INTERFACE I_EventReactionTcEvents EXTENDS I_EventReaction

METHOD GetHighestActiveEventSeverity : TcEventSeverity
END_METHOD

END_INTERFACE

(* stored: Version 1.1.0.1, ProductVersion 3.1.4026.18
   Itf I_EventReactionTcEvents: Id {9ba85094-bdcc-4410-92fb-9d3383e4ff12}
   Method GetHighestActiveEventSeverity: Id {472bb527-7b81-40a7-b14e-172cd6ea18e1} *)
